(* PLC project Unnamed, Unknown Unnamed 1 *)
(* stored: creationDateTime 2025-11-05T10:16:07, modificationDateTime 2025-11-05T10:33:59 *)

PROGRAM main
  VAR
    Sequence_Start : BOOL := False;
    Sequence_End : BOOL := False;
    Step1 : BOOL := False;
    Step1_EndCondition : BOOL := False;
    Step1_End : BOOL := False;
    Step2 : BOOL := False;
    Step2_EndCondition : BOOL := False;
    Step2_End : BOOL := False;
  END_VAR

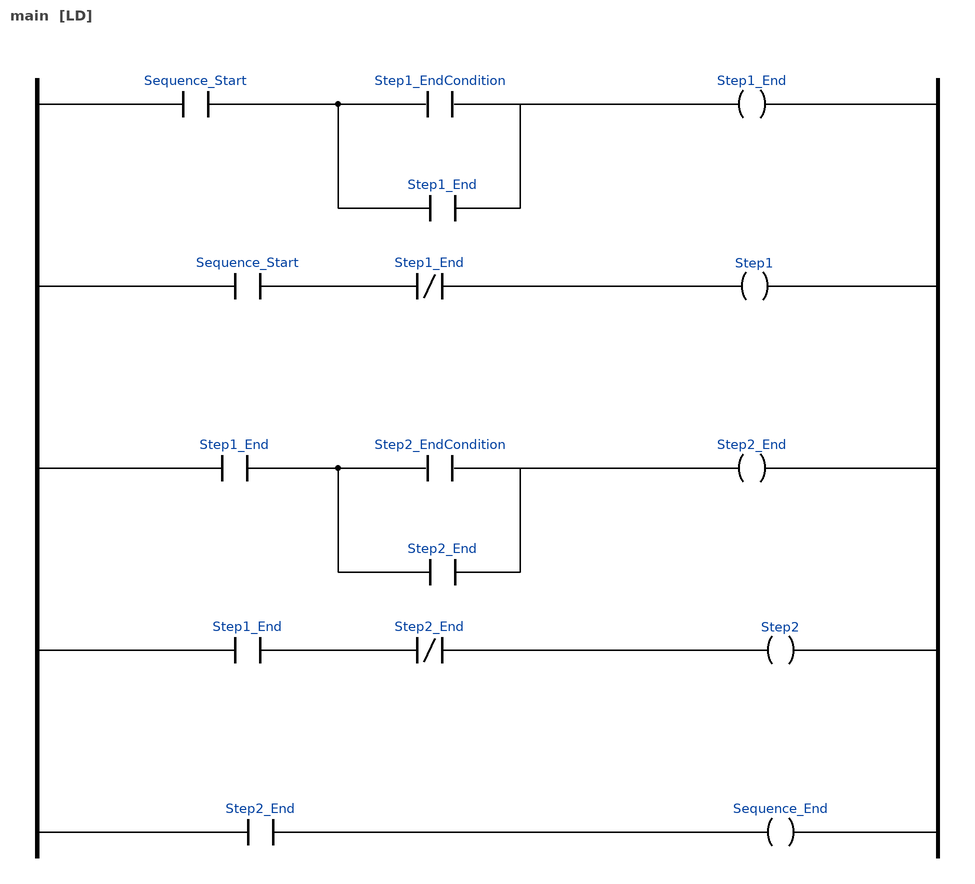
(* LD diagram, written out as Structured Text *)
Step1_End := Sequence_Start AND (Step1_EndCondition OR Step1_End);
Step1 := Sequence_Start AND NOT Step1_End;
Step2_End := Step1_End AND (Step2_EndCondition OR Step2_End);
Step2 := Step1_End AND NOT Step2_End;
Sequence_End := Step2_End;
END_PROGRAM

CONFIGURATION Config0
  RESOURCE Res0 ON PLC
    TASK task0(INTERVAL := T#20ms, PRIORITY := 0);
    PROGRAM instance0 WITH task0 : main;
  END_RESOURCE
END_CONFIGURATION
